// TIA Portal V19 export
FUNCTION "CallSimulation" : Void   // FC14, LAD
TITLE = CallSimulation
AUTHOR : Siemens Digital Industries
// This blocks switches between simulation with SIMIT and PLCSIM Advanced or with PLCSIM and PLC internal simulation function blocks
// stored: IsIECCheckEnabled true, SetENOAutomatically true
BEGIN

REGION Network 1: SIMIT simulation currently running
   // The input "0.000CC1-KE50_I1.6_SimitRunning" is a life bit from SIMIT, which is always TRUE while SIMIT is running. The following actions are performed in that case:
   // - Simulation button in HMI is not shown when a SIMIT simulation is currently running
   // - Deactivate PLC internal simulation while SIMIT simulation is running
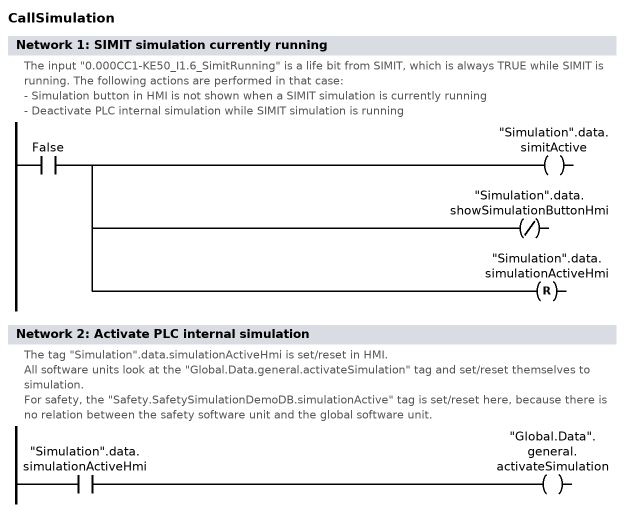
   RUNG wire#powerrail
      Contact( False )
      wire#w1
      Coil( "Simulation".data.simitActive )
   END_RUNG
   RUNG wire#w1
      I_Coil( "Simulation".data.showSimulationButtonHmi )
   END_RUNG
   RUNG wire#w1
      R_Coil( "Simulation".data.simulationActiveHmi )
   END_RUNG
   // the same network as SCL:
   "Simulation".data.simitActive := False;
   "Simulation".data.showSimulationButtonHmi := NOT False;
   IF False THEN "Simulation".data.simulationActiveHmi := FALSE; END_IF;
END_REGION

REGION Network 2: Activate PLC internal simulation
   // The tag "Simulation".data.simulationActiveHmi is set/reset in HMI.
   // 
   // All software units look at the "Global.Data.general.activateSimulation" tag and set/reset themselves to simulation.
   // 
   // For safety, the "Safety.SafetySimulationDemoDB.simulationActive" tag is set/reset here, because there is no relation between the safety software unit and the global software unit.
   RUNG wire#powerrail
      Contact( "Simulation".data.simulationActiveHmi )
      Coil( "Global.Data".general.activateSimulation )
   END_RUNG
   // the same network as SCL:
   "Global.Data".general.activateSimulation := "Simulation".data.simulationActiveHmi;
END_REGION
END_FUNCTION
